SYSTEM PNP_MVCDM (* Mechatronic Pick & Place Model/View/Diagnostics *)
  (* Standard: IEC 61499; Classification: Simulation; ApplicationDomain: Assembly; Function: Control/Diagnostics; Type: Pick & Place; Description: Mechatronic Configuration *)
  (* Version 0.6, 2008-02-18, JHC, Holobloc Inc, Moved PNP_ACT socket to 225.0.0.2:1026. *)
  (* Version 0.5, 2007-11-08, JHC, Holobloc Inc, Moved MAGNET socket from 1027 to 1036. *)
  (* Version 0.4, 2007-10-05, JHC, Holobloc Inc, Moved TAGS to end position in devices; also HMI is in last position among devices. *)
  (* Version 0.3, 2007-10-04, JHC, Holobloc Inc, Converted to Tagged Data. *)
  (* Version 0.2, 2007-09-28, JHC, Holobloc Inc, Added CNV.CLOCK.DLY, simplified PNP.CLOCK. *)
  (* Version 0.1, 2006-09-19, JHC, Holobloc Inc, Added PNP.AUTO_CTL.AUTO_GATE. *)
  (* Version 0.0, 2006-07-09, JHC, Holobloc Inc *)
  DEVICE CNV : RMT_FRAME(MGR_ID := "localhost:61500", BOUNDS := [400,100,35,180]) (* Mechatronic Conveyor Simulation *)
    RESOURCE MGR : RMT_RES
    END_RESOURCE
    RESOURCE CLOCK : EMB_RES
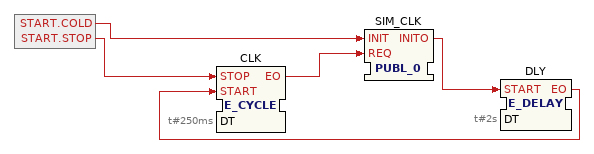
      FBS
        CLK : E_CYCLE(DT := t#250ms);
        SIM_CLK : PUBL_0; (* Simulation Clock *)
        DLY : E_DELAY(DT := t#2s); (* Wait for MODEL, VIEW initialization *)
      END_FBS
      EVENT_CONNECTIONS
        START.COLD TO SIM_CLK.INIT;
        START.STOP TO CLK.STOP;
        CLK.EO TO SIM_CLK.REQ;
        SIM_CLK.INITO TO DLY.START;
        DLY.EO TO CLK.START;
      END_CONNECTIONS
    END_RESOURCE
    RESOURCE MODEL : EMB_RES
      FBS
        CNV : CNV_MDLL(VF := 10, ACT_ID := "CNV_MTR_AUTO");
        PRESENT : PUBL_1; (* Workpiece present at end of conveyor *)
        S0_SENSE : V_SENSE(REFSTYLE := VSTYLE#BALL);
        CNV_UNLD : SUBL_0;
      END_FBS
      EVENT_CONNECTIONS
        CNV.INDS TO S0_SENSE.SENSE;
        S0_SENSE.IND TO PRESENT.REQ;
        CNV.INITO TO PRESENT.INIT;
        START.COLD TO CNV_UNLD.INIT;
        CNV_UNLD.INITO TO CNV.INIT;
        CNV_UNLD.IND TO CNV.UNLD;
      END_CONNECTIONS
      DATA_CONNECTIONS
        CNV.END TO S0_SENSE.PRESENT;
        CNV.STYLO TO S0_SENSE.STYLE;
        S0_SENSE.Q TO PRESENT.SD_1;
      END_CONNECTIONS
    END_RESOURCE
    RESOURCE VIEW : VIEW_PANEL(DIA := 25, SIZE := [1,5])
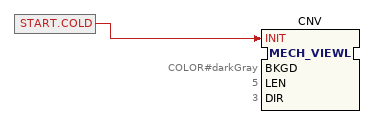
      FBS
        CNV : MECH_VIEWL(BKGD := COLOR#darkGray, LEN := 5, DIR := 3); (* Conveyor *)
      END_FBS
      EVENT_CONNECTIONS
        START.COLD TO CNV.INIT;
      END_CONNECTIONS
    END_RESOURCE
    RESOURCE CTL : EMB_RES (* Conveyor Control *)
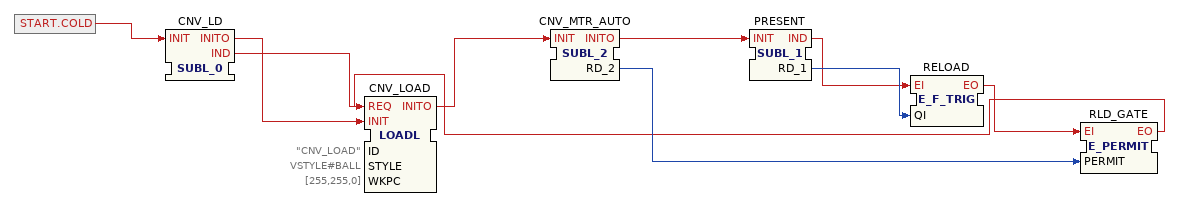
      FBS
        CNV_LOAD : LOADL(ID := "CNV_LOAD", STYLE := VSTYLE#BALL, WKPC := [255,255,0]);
        CNV_MTR_AUTO : SUBL_2; (* Conveyor MOTOR and AUTO signals from HMI *)
        PRESENT : SUBL_1; (* Workpiece present at end of conveyor *)
        RELOAD : E_F_TRIG;
        RLD_GATE : E_PERMIT;
        CNV_LD : SUBL_0;
      END_FBS
      EVENT_CONNECTIONS
        CNV_LOAD.INITO TO CNV_MTR_AUTO.INIT;
        RELOAD.EO TO RLD_GATE.EI;
        RLD_GATE.EO TO CNV_LOAD.REQ;
        START.COLD TO CNV_LD.INIT;
        CNV_LD.INITO TO CNV_LOAD.INIT;
        CNV_LD.IND TO CNV_LOAD.REQ;
        PRESENT.IND TO RELOAD.EI;
        CNV_MTR_AUTO.INITO TO PRESENT.INIT;
      END_CONNECTIONS
      DATA_CONNECTIONS
        PRESENT.RD_1 TO RELOAD.QI;
        CNV_MTR_AUTO.RD_2 TO RLD_GATE.PERMIT;
      END_CONNECTIONS
    END_RESOURCE
    RESOURCE TAGS : EMB_RES
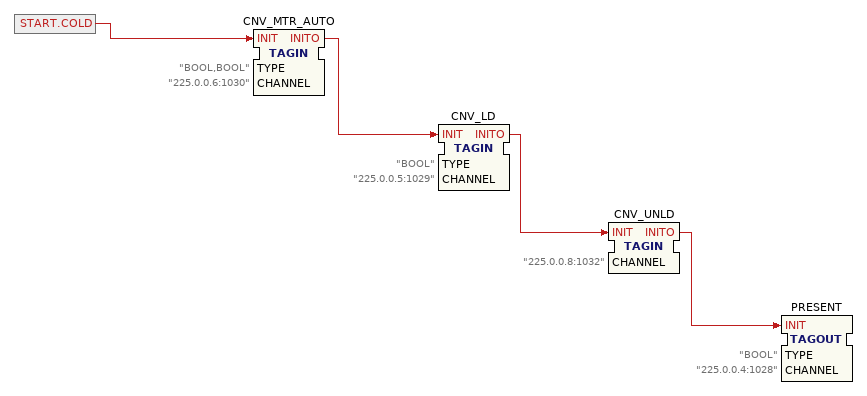
      FBS
        CNV_MTR_AUTO : TAGIN(TYPE := "BOOL,BOOL", CHANNEL := "225.0.0.6:1030");
        CNV_LD : TAGIN(TYPE := "BOOL", CHANNEL := "225.0.0.5:1029"); (* Remote LOAD Command to Conveyor *)
        CNV_UNLD : TAGIN(CHANNEL := "225.0.0.8:1032");
        PRESENT : TAGOUT(TYPE := "BOOL", CHANNEL := "225.0.0.4:1028"); (* Workpiece present at end of conveyor *)
      END_FBS
      EVENT_CONNECTIONS
        START.COLD TO CNV_MTR_AUTO.INIT;
        CNV_MTR_AUTO.INITO TO CNV_LD.INIT;
        CNV_LD.INITO TO CNV_UNLD.INIT;
        CNV_UNLD.INITO TO PRESENT.INIT;
      END_CONNECTIONS
    END_RESOURCE
  END_DEVICE
  DEVICE PNP : RMT_FRAME(BOUNDS := [430,100,135,180]) (* Mechatronic two-dimensional Pick&Place Unit *)
    RESOURCE MGR : RMT_RES
    END_RESOURCE
    RESOURCE CLOCK : EMB_RES
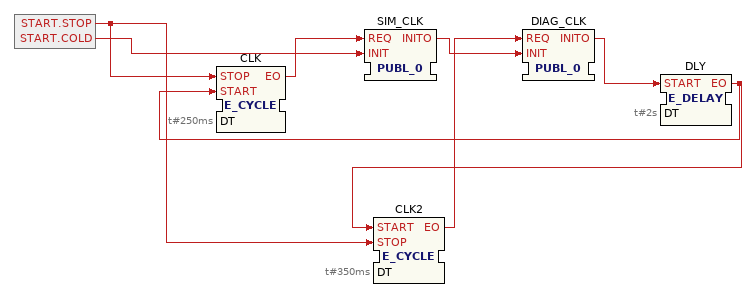
      FBS
        CLK : E_CYCLE(DT := t#250ms);
        SIM_CLK : PUBL_0; (* Simulation Clock *)
        CLK2 : E_CYCLE(DT := t#350ms);
        DIAG_CLK : PUBL_0; (* Diagnostics Clock *)
        DLY : E_DELAY(DT := t#2s); (* Wait for MODEL, VIEW initialization *)
      END_FBS
      EVENT_CONNECTIONS
        START.STOP TO CLK.STOP;
        CLK2.EO TO DIAG_CLK.REQ;
        CLK.EO TO SIM_CLK.REQ;
        START.COLD TO SIM_CLK.INIT;
        SIM_CLK.INITO TO DIAG_CLK.INIT;
        DIAG_CLK.INITO TO DLY.START;
        DLY.EO TO CLK.START;
        DLY.EO TO CLK2.START;
        START.STOP TO CLK2.STOP;
      END_CONNECTIONS
    END_RESOURCE
    RESOURCE XY : EMB_RES
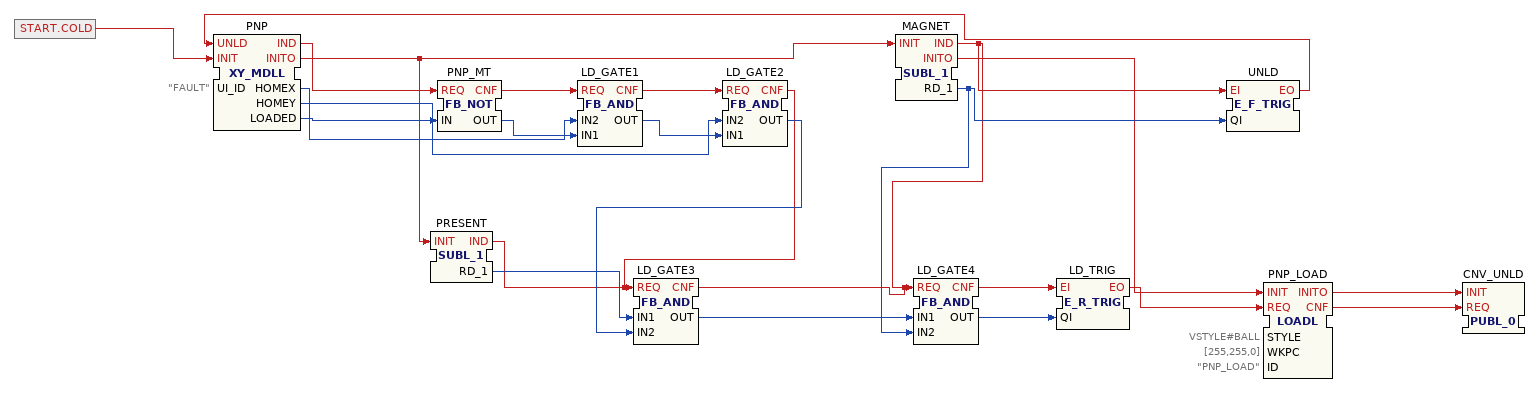
      FBS
        PNP : XY_MDLL(UI_ID := "FAULT");
        MAGNET : SUBL_1; (* PICK magnet actuation *)
        LD_GATE1 : FB_AND;
        CNV_UNLD : PUBL_0;
        PNP_MT : FB_NOT; (* No workpiece loaded to PNP unit *)
        LD_GATE2 : FB_AND;
        UNLD : E_F_TRIG;
        PRESENT : SUBL_1;
        LD_GATE3 : FB_AND;
        LD_GATE4 : FB_AND;
        LD_TRIG : E_R_TRIG;
        PNP_LOAD : LOADL(STYLE := VSTYLE#BALL, WKPC := [255,255,0], ID := "PNP_LOAD");
      END_FBS
      EVENT_CONNECTIONS
        MAGNET.IND TO UNLD.EI;
        UNLD.EO TO PNP.UNLD;
        PNP.IND TO PNP_MT.REQ;
        PNP_MT.CNF TO LD_GATE1.REQ;
        LD_GATE1.CNF TO LD_GATE2.REQ;
        PRESENT.IND TO LD_GATE3.REQ;
        MAGNET.IND TO LD_GATE4.REQ;
        LD_GATE3.CNF TO LD_GATE4.REQ;
        LD_GATE4.CNF TO LD_TRIG.EI;
        START.COLD TO PNP.INIT;
        MAGNET.INITO TO PNP_LOAD.INIT;
        LD_TRIG.EO TO PNP_LOAD.REQ;
        PNP_LOAD.INITO TO CNV_UNLD.INIT;
        PNP_LOAD.CNF TO CNV_UNLD.REQ;
        LD_GATE2.CNF TO LD_GATE3.REQ;
        PNP.INITO TO MAGNET.INIT;
        PNP.INITO TO PRESENT.INIT;
      END_CONNECTIONS
      DATA_CONNECTIONS
        MAGNET.RD_1 TO UNLD.QI;
        PNP.HOMEX TO LD_GATE1.IN2;
        PNP.HOMEY TO LD_GATE2.IN2;
        LD_GATE1.OUT TO LD_GATE2.IN1;
        PRESENT.RD_1 TO LD_GATE3.IN1;
        LD_GATE2.OUT TO LD_GATE3.IN2;
        LD_GATE4.OUT TO LD_TRIG.QI;
        PNP.LOADED TO PNP_MT.IN;
        PNP_MT.OUT TO LD_GATE1.IN1;
        LD_GATE3.OUT TO LD_GATE4.IN1;
        MAGNET.RD_1 TO LD_GATE4.IN2;
      END_CONNECTIONS
    END_RESOURCE
    RESOURCE VIEW : VIEW_PANEL(DIA := 25, SIZE := [5,5], VERTICAL := 0)
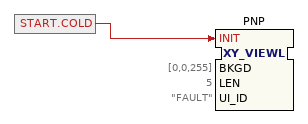
      FBS
        PNP : XY_VIEWL(BKGD := [0,0,255], LEN := 5, UI_ID := "FAULT");
      END_FBS
      EVENT_CONNECTIONS
        START.COLD TO PNP.INIT;
      END_CONNECTIONS
    END_RESOURCE
    RESOURCE DIAGNOSTICS : EMB_RES
      FBS
        PNP_ACT : SUBL_4;
        PNP_SENSE : SUBL_5;
        X_FWD : MECH1_DIAGL(N := 10, SRC := "X-AXIS", MSG := "TIMEOUT ADVANCING");
        X_REV : MECH1_DIAGL(N := 10, SRC := "X_AXIS", MSG := "TIMEOUT RETRACTING");
        Y_FWD : MECH1_DIAGL(N := 10, SRC := "Y-AXIS", MSG := "TIMEOUT ADVANCING");
        Y_REV : MECH1_DIAGL(N := 10, SRC := "Y-AXIS", MSG := "TIMEOUT RETRACTING");
      END_FBS
      EVENT_CONNECTIONS
        X_FWD.INITO TO X_REV.INIT;
        X_REV.INITO TO Y_FWD.INIT;
        Y_FWD.INITO TO Y_REV.INIT;
        START.COLD TO X_FWD.INIT;
        Y_REV.INITO TO PNP_ACT.INIT;
        PNP_ACT.INITO TO PNP_SENSE.INIT;
      END_CONNECTIONS
      DATA_CONNECTIONS
        PNP_ACT.RD_1 TO X_FWD.FWD;
        PNP_SENSE.RD_3 TO X_FWD.END;
        PNP_ACT.RD_2 TO X_REV.FWD;
        PNP_SENSE.RD_2 TO X_REV.END;
        PNP_ACT.RD_3 TO Y_FWD.FWD;
        PNP_SENSE.RD_5 TO Y_FWD.END;
        PNP_ACT.RD_4 TO Y_REV.FWD;
        PNP_SENSE.RD_4 TO Y_REV.END;
      END_CONNECTIONS
    END_RESOURCE
    RESOURCE AUTO_CTL : EMB_RES
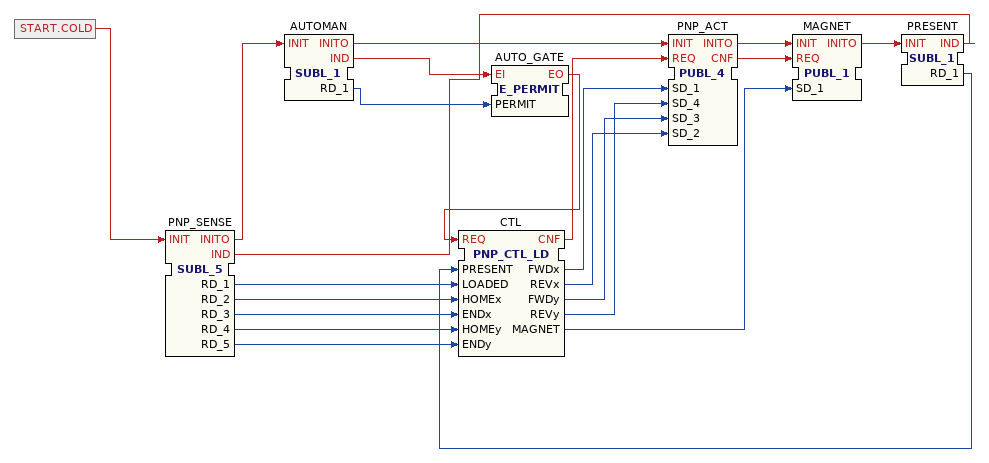
      FBS
        CTL : PNP_CTL_LD;
        AUTOMAN : SUBL_1;
        MAGNET : PUBL_1;
        PNP_ACT : PUBL_4; (* Actuators to PNP unit *)
        PNP_SENSE : SUBL_5; (* Sensors from PNP unit *)
        PRESENT : SUBL_1;
        AUTO_GATE : E_PERMIT;
      END_FBS
      EVENT_CONNECTIONS
        START.COLD TO PNP_SENSE.INIT;
        AUTOMAN.INITO TO PNP_ACT.INIT;
        CTL.CNF TO PNP_ACT.REQ;
        PNP_ACT.INITO TO MAGNET.INIT;
        PNP_ACT.CNF TO MAGNET.REQ;
        MAGNET.INITO TO PRESENT.INIT;
        PNP_SENSE.INITO TO AUTOMAN.INIT;
        AUTOMAN.IND TO AUTO_GATE.EI;
        PRESENT.IND TO AUTO_GATE.EI;
        PNP_SENSE.IND TO AUTO_GATE.EI;
        AUTO_GATE.EO TO CTL.REQ;
      END_CONNECTIONS
      DATA_CONNECTIONS
        CTL.MAGNET TO MAGNET.SD_1;
        CTL.FWDx TO PNP_ACT.SD_1;
        CTL.REVy TO PNP_ACT.SD_4;
        CTL.FWDy TO PNP_ACT.SD_3;
        CTL.REVx TO PNP_ACT.SD_2;
        PRESENT.RD_1 TO CTL.PRESENT;
        PNP_SENSE.RD_1 TO CTL.LOADED;
        PNP_SENSE.RD_2 TO CTL.HOMEx;
        PNP_SENSE.RD_3 TO CTL.ENDx;
        PNP_SENSE.RD_4 TO CTL.HOMEy;
        PNP_SENSE.RD_5 TO CTL.ENDy;
        AUTOMAN.RD_1 TO AUTO_GATE.PERMIT;
      END_CONNECTIONS
    END_RESOURCE
    RESOURCE TAGS : EMB_RES
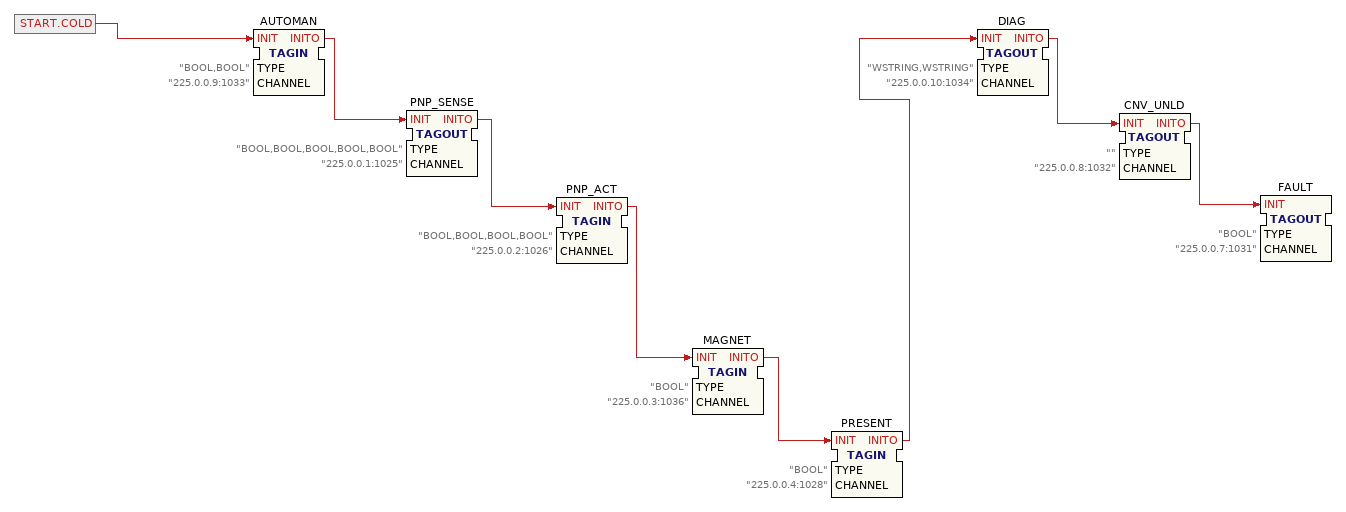
      FBS
        PNP_ACT : TAGIN(TYPE := "BOOL,BOOL,BOOL,BOOL", CHANNEL := "225.0.0.2:1026");
        PNP_SENSE : TAGOUT(TYPE := "BOOL,BOOL,BOOL,BOOL,BOOL", CHANNEL := "225.0.0.1:1025"); (* Sensors from PNP unit *)
        DIAG : TAGOUT(TYPE := "WSTRING,WSTRING", CHANNEL := "225.0.0.10:1034"); (* Diagnostic SRC(source)+COND(ition) data *)
        AUTOMAN : TAGIN(TYPE := "BOOL,BOOL", CHANNEL := "225.0.0.9:1033"); (* PNP AUTO+MANUAL modes *)
        MAGNET : TAGIN(TYPE := "BOOL", CHANNEL := "225.0.0.3:1036");
        PRESENT : TAGIN(TYPE := "BOOL", CHANNEL := "225.0.0.4:1028"); (* Workpiece present at end of conveyor *)
        CNV_UNLD : TAGOUT(TYPE := "", CHANNEL := "225.0.0.8:1032"); (* Simulation event to unload piece from conveyor *)
        FAULT : TAGOUT(TYPE := "BOOL", CHANNEL := "225.0.0.7:1031"); (* Motor overload fault sensor *)
      END_FBS
      EVENT_CONNECTIONS
        PNP_SENSE.INITO TO PNP_ACT.INIT;
        START.COLD TO AUTOMAN.INIT;
        AUTOMAN.INITO TO PNP_SENSE.INIT;
        PNP_ACT.INITO TO MAGNET.INIT;
        MAGNET.INITO TO PRESENT.INIT;
        PRESENT.INITO TO DIAG.INIT;
        DIAG.INITO TO CNV_UNLD.INIT;
        CNV_UNLD.INITO TO FAULT.INIT;
      END_CONNECTIONS
    END_RESOURCE
  END_DEVICE
  DEVICE HMI : FRAME_DEVICE(BOUNDS := [100,100,300,180], GRID := [1,4])
    RESOURCE CONVEYOR : PANEL_RESOURCE
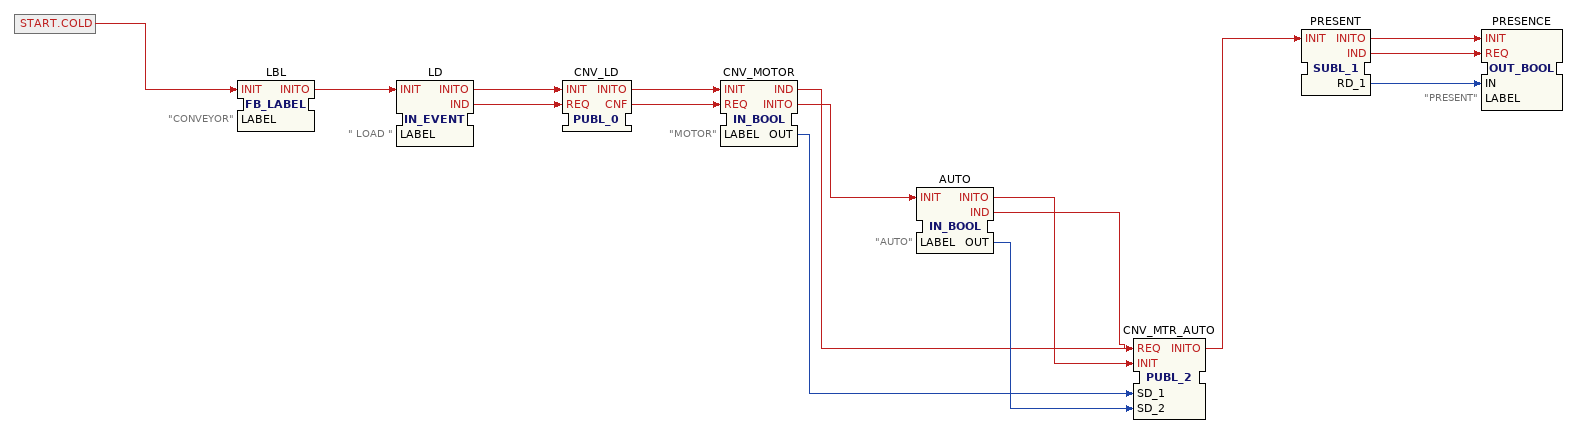
      FBS
        LD : IN_EVENT(LABEL := "    LOAD    ");
        CNV_LD : PUBL_0;
        CNV_MOTOR : IN_BOOL(LABEL := "MOTOR");
        CNV_MTR_AUTO : PUBL_2;
        PRESENT : SUBL_1; (* Workpiece present at end of conveyor *)
        AUTO : IN_BOOL(LABEL := "AUTO"); (* Conveyor auto-reload *)
        LBL : FB_LABEL(LABEL := "CONVEYOR");
        PRESENCE : OUT_BOOL(LABEL := "PRESENT");
      END_FBS
      EVENT_CONNECTIONS
        LD.INITO TO CNV_LD.INIT;
        LD.IND TO CNV_LD.REQ;
        CNV_LD.INITO TO CNV_MOTOR.INIT;
        CNV_LD.CNF TO CNV_MOTOR.REQ;
        CNV_MOTOR.IND TO CNV_MTR_AUTO.REQ;
        START.COLD TO LBL.INIT;
        LBL.INITO TO LD.INIT;
        PRESENT.INITO TO PRESENCE.INIT;
        PRESENT.IND TO PRESENCE.REQ;
        CNV_MOTOR.INITO TO AUTO.INIT;
        AUTO.INITO TO CNV_MTR_AUTO.INIT;
        AUTO.IND TO CNV_MTR_AUTO.REQ;
        CNV_MTR_AUTO.INITO TO PRESENT.INIT;
      END_CONNECTIONS
      DATA_CONNECTIONS
        CNV_MOTOR.OUT TO CNV_MTR_AUTO.SD_1;
        PRESENT.RD_1 TO PRESENCE.IN;
        AUTO.OUT TO CNV_MTR_AUTO.SD_2;
      END_CONNECTIONS
    END_RESOURCE
    RESOURCE MODE_CTL : PANEL_RESOURCE
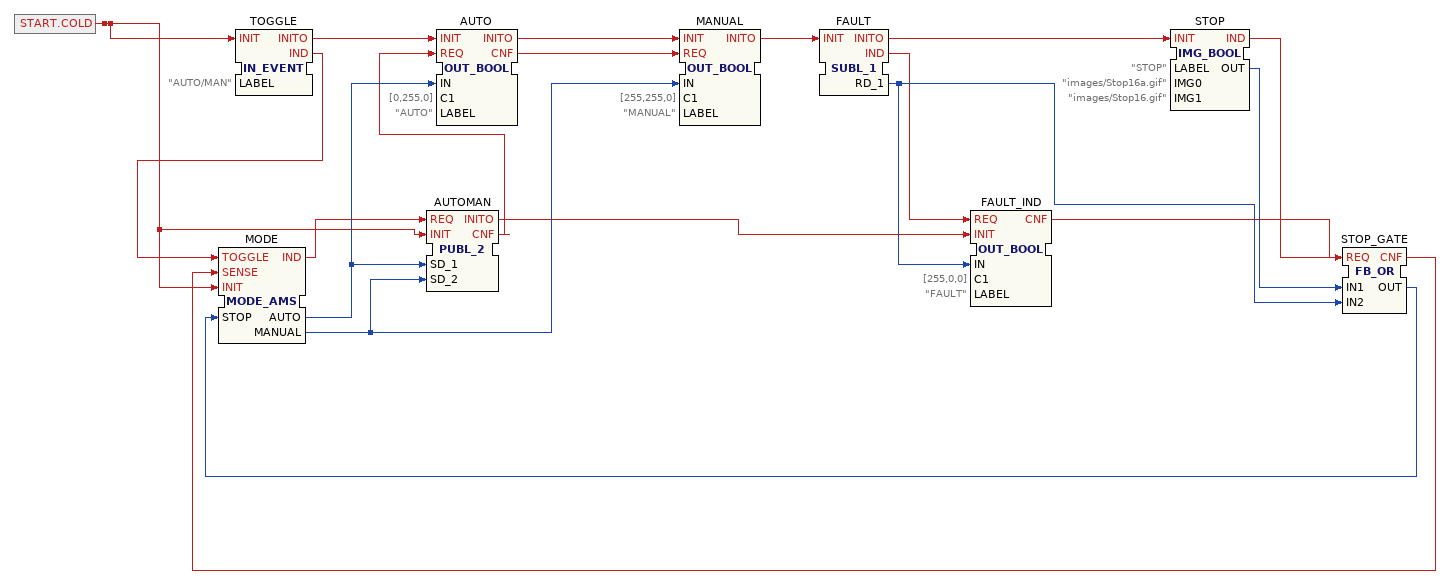
      FBS
        FAULT_IND : OUT_BOOL(C1 := [255,0,0], LABEL := "FAULT");
        FAULT : SUBL_1; (* Motor overload fault sensor *)
        AUTOMAN : PUBL_2;
        MODE : MODE_AMS;
        TOGGLE : IN_EVENT(LABEL := "AUTO/MAN");
        AUTO : OUT_BOOL(C1 := [0,255,0], LABEL := "AUTO");
        MANUAL : OUT_BOOL(C1 := [255,255,0], LABEL := "MANUAL");
        STOP : IMG_BOOL(LABEL := "STOP", IMG0 := "images/Stop16a.gif", IMG1 := "images/Stop16.gif");
        STOP_GATE : FB_OR;
      END_FBS
      EVENT_CONNECTIONS
        START.COLD TO TOGGLE.INIT;
        TOGGLE.INITO TO AUTO.INIT;
        AUTO.INITO TO MANUAL.INIT;
        AUTO.CNF TO MANUAL.REQ;
        MODE.IND TO AUTOMAN.REQ;
        TOGGLE.IND TO MODE.TOGGLE;
        STOP.IND TO STOP_GATE.REQ;
        MANUAL.INITO TO FAULT.INIT;
        FAULT.INITO TO STOP.INIT;
        FAULT.IND TO FAULT_IND.REQ;
        FAULT_IND.CNF TO STOP_GATE.REQ;
        STOP_GATE.CNF TO MODE.SENSE;
        START.COLD TO AUTOMAN.INIT;
        START.COLD TO MODE.INIT;
        AUTOMAN.INITO TO FAULT_IND.INIT;
        AUTOMAN.CNF TO AUTO.REQ;
      END_CONNECTIONS
      DATA_CONNECTIONS
        FAULT.RD_1 TO FAULT_IND.IN;
        MODE.AUTO TO AUTOMAN.SD_1;
        MODE.MANUAL TO AUTOMAN.SD_2;
        MODE.AUTO TO AUTO.IN;
        MODE.MANUAL TO MANUAL.IN;
        STOP.OUT TO STOP_GATE.IN1;
        FAULT.RD_1 TO STOP_GATE.IN2;
        STOP_GATE.OUT TO MODE.STOP;
      END_CONNECTIONS
    END_RESOURCE
    RESOURCE ACTUATORS : PANEL_RESOURCE
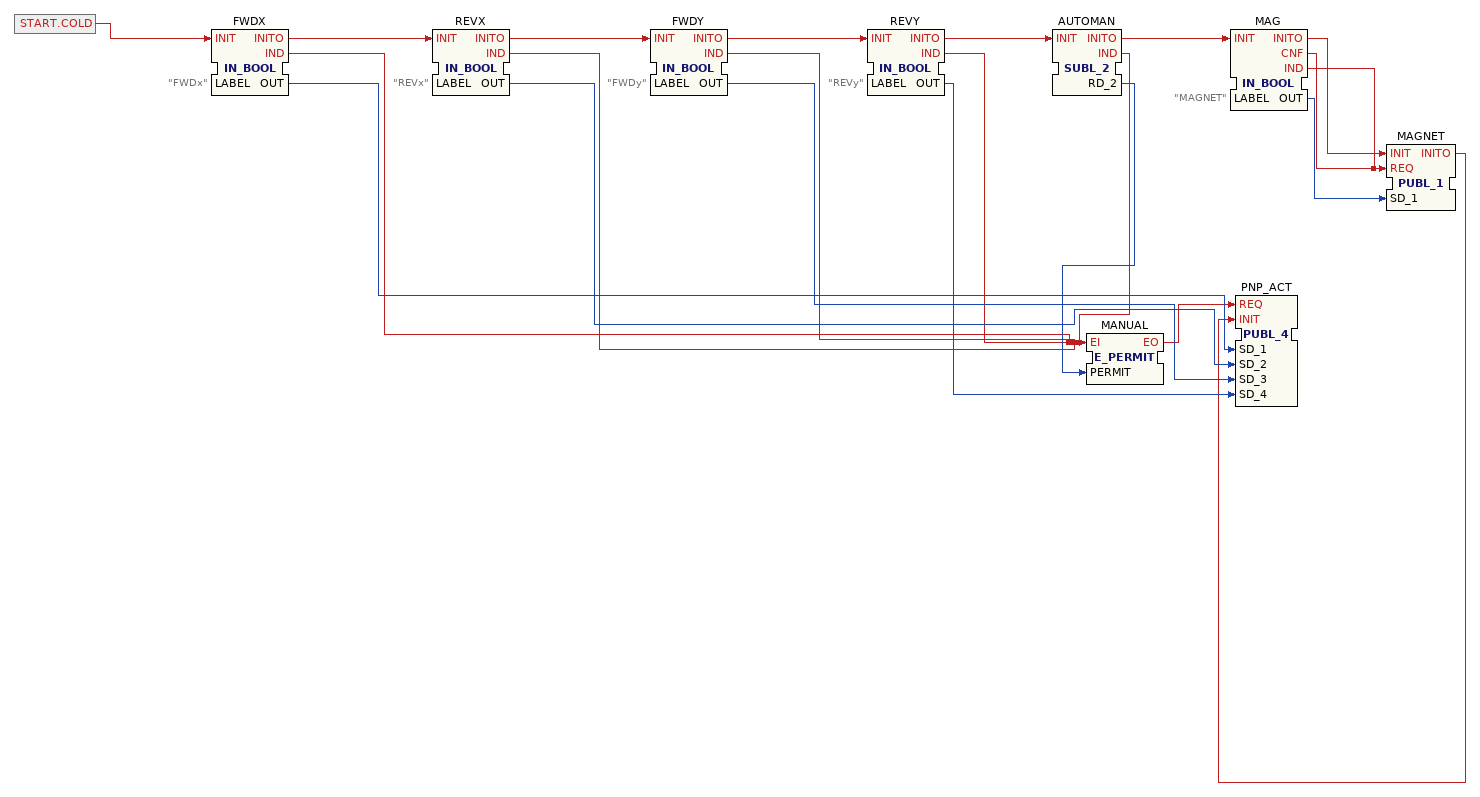
      FBS
        PNP_ACT : PUBL_4;
        FWDX : IN_BOOL(LABEL := "FWDx");
        REVX : IN_BOOL(LABEL := "REVx");
        FWDY : IN_BOOL(LABEL := "FWDy");
        REVY : IN_BOOL(LABEL := "REVy");
        MAG : IN_BOOL(LABEL := "MAGNET");
        MAGNET : PUBL_1;
        AUTOMAN : SUBL_2;
        MANUAL : E_PERMIT;
      END_FBS
      EVENT_CONNECTIONS
        START.COLD TO FWDX.INIT;
        FWDX.INITO TO REVX.INIT;
        REVX.INITO TO FWDY.INIT;
        FWDY.INITO TO REVY.INIT;
        MAG.INITO TO MAGNET.INIT;
        MAG.CNF TO MAGNET.REQ;
        MAG.IND TO MAGNET.REQ;
        REVY.INITO TO AUTOMAN.INIT;
        MANUAL.EO TO PNP_ACT.REQ;
        REVY.IND TO MANUAL.EI;
        FWDY.IND TO MANUAL.EI;
        REVX.IND TO MANUAL.EI;
        FWDX.IND TO MANUAL.EI;
        AUTOMAN.INITO TO MAG.INIT;
        MAGNET.INITO TO PNP_ACT.INIT;
        AUTOMAN.IND TO MANUAL.EI;
      END_CONNECTIONS
      DATA_CONNECTIONS
        FWDX.OUT TO PNP_ACT.SD_1;
        REVX.OUT TO PNP_ACT.SD_2;
        FWDY.OUT TO PNP_ACT.SD_3;
        REVY.OUT TO PNP_ACT.SD_4;
        MAG.OUT TO MAGNET.SD_1;
        AUTOMAN.RD_2 TO MANUAL.PERMIT;
      END_CONNECTIONS
    END_RESOURCE
    RESOURCE SENSORS : PANEL_RESOURCE
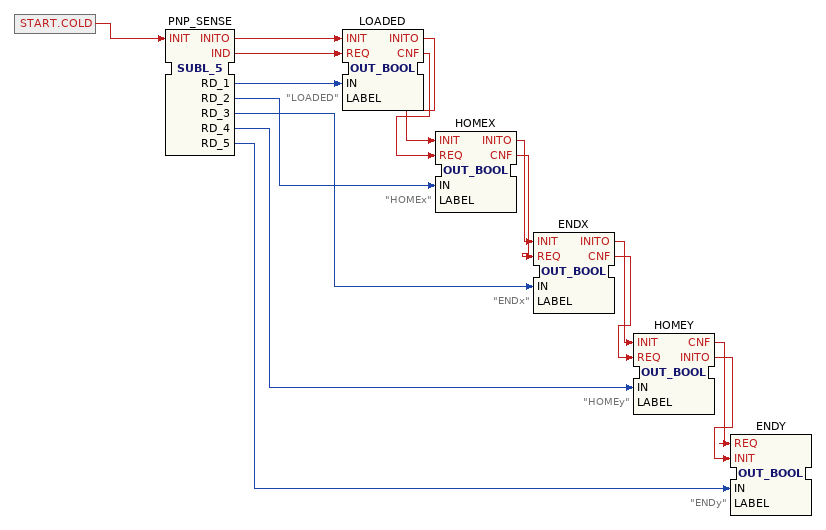
      FBS
        PNP_SENSE : SUBL_5;
        HOMEX : OUT_BOOL(LABEL := "HOMEx");
        ENDX : OUT_BOOL(LABEL := "ENDx");
        HOMEY : OUT_BOOL(LABEL := "HOMEy");
        ENDY : OUT_BOOL(LABEL := "ENDy");
        LOADED : OUT_BOOL(LABEL := "LOADED");
      END_FBS
      EVENT_CONNECTIONS
        START.COLD TO PNP_SENSE.INIT;
        HOMEX.INITO TO ENDX.INIT;
        HOMEX.CNF TO ENDX.REQ;
        ENDX.INITO TO HOMEY.INIT;
        HOMEY.CNF TO ENDY.REQ;
        HOMEY.INITO TO ENDY.INIT;
        ENDX.CNF TO HOMEY.REQ;
        PNP_SENSE.INITO TO LOADED.INIT;
        LOADED.INITO TO HOMEX.INIT;
        PNP_SENSE.IND TO LOADED.REQ;
        LOADED.CNF TO HOMEX.REQ;
      END_CONNECTIONS
      DATA_CONNECTIONS
        PNP_SENSE.RD_1 TO LOADED.IN;
        PNP_SENSE.RD_2 TO HOMEX.IN;
        PNP_SENSE.RD_3 TO ENDX.IN;
        PNP_SENSE.RD_4 TO HOMEY.IN;
        PNP_SENSE.RD_5 TO ENDY.IN;
      END_CONNECTIONS
    END_RESOURCE
    RESOURCE TAGS : EMB_RES
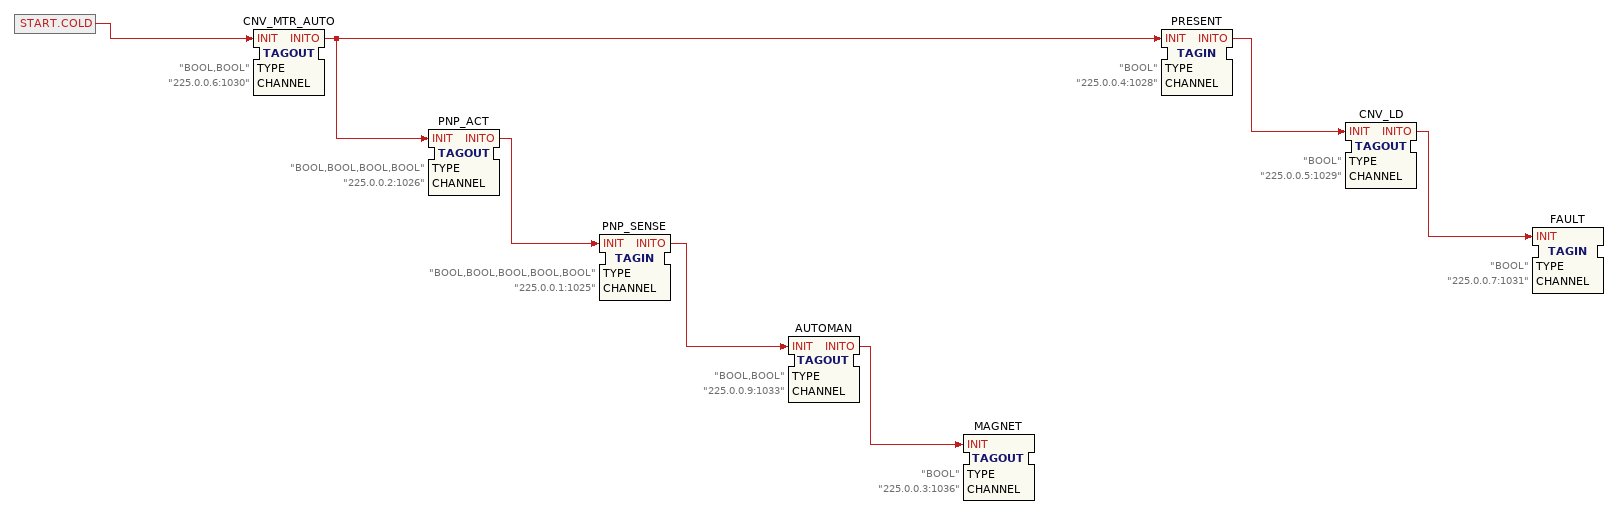
      FBS
        CNV_MTR_AUTO : TAGOUT(TYPE := "BOOL,BOOL", CHANNEL := "225.0.0.6:1030");
        PNP_ACT : TAGOUT(TYPE := "BOOL,BOOL,BOOL,BOOL", CHANNEL := "225.0.0.2:1026");
        PNP_SENSE : TAGIN(TYPE := "BOOL,BOOL,BOOL,BOOL,BOOL", CHANNEL := "225.0.0.1:1025");
        AUTOMAN : TAGOUT(TYPE := "BOOL,BOOL", CHANNEL := "225.0.0.9:1033");
        MAGNET : TAGOUT(TYPE := "BOOL", CHANNEL := "225.0.0.3:1036");
        PRESENT : TAGIN(TYPE := "BOOL", CHANNEL := "225.0.0.4:1028");
        CNV_LD : TAGOUT(TYPE := "BOOL", CHANNEL := "225.0.0.5:1029");
        FAULT : TAGIN(TYPE := "BOOL", CHANNEL := "225.0.0.7:1031"); (* Motor overload fault sensor *)
      END_FBS
      EVENT_CONNECTIONS
        START.COLD TO CNV_MTR_AUTO.INIT;
        CNV_MTR_AUTO.INITO TO PNP_ACT.INIT;
        PNP_ACT.INITO TO PNP_SENSE.INIT;
        PNP_SENSE.INITO TO AUTOMAN.INIT;
        AUTOMAN.INITO TO MAGNET.INIT;
        CNV_MTR_AUTO.INITO TO PRESENT.INIT;
        PRESENT.INITO TO CNV_LD.INIT;
        CNV_LD.INITO TO FAULT.INIT;
      END_CONNECTIONS
    END_RESOURCE
  END_DEVICE
  DEVICE DIAGNOSTICS : FRAME_DEVICE(BOUNDS := [100,280,450,180])
    RESOURCE LOG : PANEL_RESOURCE(ROWS := 1, COLS := 1)
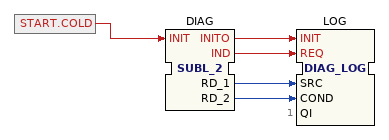
      FBS
        DIAG : SUBL_2;
        LOG : DIAG_LOG(QI := 1);
      END_FBS
      EVENT_CONNECTIONS
        START.COLD TO DIAG.INIT;
        DIAG.INITO TO LOG.INIT;
        DIAG.IND TO LOG.REQ;
      END_CONNECTIONS
      DATA_CONNECTIONS
        DIAG.RD_1 TO LOG.SRC;
        DIAG.RD_2 TO LOG.COND;
      END_CONNECTIONS
    END_RESOURCE
    RESOURCE TAGS : EMB_RES
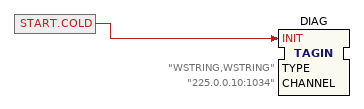
      FBS
        DIAG : TAGIN(TYPE := "WSTRING,WSTRING", CHANNEL := "225.0.0.10:1034");
      END_FBS
      EVENT_CONNECTIONS
        START.COLD TO DIAG.INIT;
      END_CONNECTIONS
    END_RESOURCE
  END_DEVICE
END_SYSTEM
